FUNCTION_BLOCK Test_TExecutionWhenReady_Start_SelectsStarting EXTENDS T_UnitTestbase
VAR
    Execution : T_Execution;
END_VAR

// Setup...
Execution.FB_init(bInitRetains := FALSE,
                  bInCopyCode  := FALSE);

// Test...
Execution.Start();

Assertion.AssertEquals_BOOL(Expected     := TRUE,
                            Actual       := Execution.Starting,
                            VariableName := 'Execution.Starting');

TestFinished();

END_FUNCTION_BLOCK

(* stored: Version 1.1.0.1, ProductVersion 3.1.4024.6
   POU Test_TExecutionWhenReady_Start_SelectsStarting: Id {ef98dc1e-565d-4e35-b9f5-21bb06b550cf}, SpecialFunc None *)
